(* IEC 61131-3 sources: eCockpitGit/test_project/src/%PLC%PLCTest2/%PLOG%Plc Logic/%APP%APP1_Test/%F%NormalFolder/%GVL%GVL_test_1/%PRO%PropAlop_1, 1 file *)

(* ---- %GETSET%Set.st ---- *)
VAR
	temp3:INT;
END_VAR

(*%!%__DELIMITER__%!%*)
variablssss1		:=		temp3 + PropAlop_1;
